// TIA Portal project "stl_demo_2" (V15)

(* hardware
DEVICE "S7-400 station_1"  S7-400 station
   slot 0: "UR1_0"  UR1  6ES7 400-1TA01-0AA0
   slot 1: "PS 405 4A_1"  PS 405 4A  6ES7 405-0DA02-0AA0
   slot 2: "PLC_1"  CPU 412-2 PN  6ES7 412-2EK07-0AB0  V7.0
      slot 2: "MPI/DP interface_1"  X1
      slot 5: "PROFINET interface_1"  PN-IO
         slot 1: "Port_1"  Port
         slot 2: "Port_2"  Port
   slot 3: "DI 32x24VDC_1"  DI32 x 24VDC  6ES7 421-1BL01-0AA0
   slot 4: "DI 16x24VDC_1"  DI16 x 24VDC interrupt  6ES7 421-7BH01-0AB0
   slot 5: "DO 16x24VDC/2A_1"  DO16 x 24VDC / 2A  6ES7 422-1BH11-0AA0
*)

// ===== PLC "PLC_1"  CPU 412-2 PN =====

VAR_GLOBAL   // PLC tag table "TAG_STL_OUT"
   "Q0.0" AT %M100.0 : Bool;
   "Q0.1" AT %M100.1 : Bool;
END_VAR

VAR_GLOBAL   // PLC tag table "tag_stl_IN"
   "M10.0" AT %M10.0 : Bool;
   "M10.1" AT %M10.1 : Bool;
   "M10.2" AT %M10.2 : Bool;
   "M10.3" AT %M10.3 : Bool;
   "M10.4" AT %M10.4 : Bool;
   "M10.5" AT %M10.5 : Bool;
   "M10.6" AT %M10.6 : Bool;
   "M10.7" AT %M10.7 : Bool;
   "M11.0" AT %M11.0 : Bool;
   "M11.1" AT %M11.1 : Bool;
   "M11.2" AT %M11.2 : Bool;
END_VAR

ORGANIZATION_BLOCK "Main"   // OB1, LAD
TITLE = "Main Program Sweep (Cycle)"
{ S7_Optimized_Access := 'FALSE' }
VERSION : 0.1
   VAR_TEMP
      OB1_EV_CLASS : Byte;   // Bits 0-3 = 1 (Coming event), Bits 4-7 = 1 (Event class 1)
      OB1_SCAN_1 : Byte;   // 1 (Cold restart scan 1 of OB 1), 3 (Scan 2-n of OB 1)
      OB1_PRIORITY : Byte;   // Priority of OB Execution
      OB1_OB_NUMBR : Byte;   // 1 (Organization block 1, OB1)
      OB1_RESERVED_1 : Byte;   // Reserved for system
      OB1_RESERVED_2 : Byte;   // Reserved for system
      OB1_PREV_CYCLE : Int;   // Cycle time of previous OB1 scan (milliseconds)
      OB1_MIN_CYCLE : Int;   // Minimum cycle time of OB1 (milliseconds)
      OB1_MAX_CYCLE : Int;   // Maximum cycle time of OB1 (milliseconds)
      OB1_DATE_TIME : Date_And_Time;   // Date and time OB1 started
   END_VAR
BEGIN

REGION Network 1 (STL)
         A(;
         O     "M10.0";
         O(;
         A     "M10.1";
         AN    "M10.2";
         );
         ON    "M10.3";
         );
   //
END_REGION
END_ORGANIZATION_BLOCK